{attribute 'qualified_only'}
VAR_GLOBAL
	Extruder		: ST_ExtruderControl;
	HeaterTop		: ST_HeaterZone;
	HeaterMiddle	: ST_HeaterZone;	
	HeaterNozzle	: ST_HeaterZone;
	ExtruderMotor	: ST_MotorControl;
END_VAR

(* stored: Version 1.1.0.1
   GVL GVL_Extruder: Id {b036e722-566c-4769-a1fd-4d2cf706f655} *)
